TEXTLIST FaultState
  0 = ' '
  1 = 'Fault'
   = ''
END_TEXTLIST

(* stored: Version 1.1.0.1, ProductVersion 3.1.4024.12
   TextList FaultState: Id {ea1b1b23-3e92-4569-b6f9-d1945a018b1c} *)
